FUNCTION_BLOCK PUBLIC ACMethodMixing EXTENDS ACMethodRouteBase
VAR_INPUT
END_VAR
VAR_OUTPUT
END_VAR
VAR PERSISTENT
	_Parameter : ACMethodMixingP;
	_Result : ACMethodMixingR;
END_VAR

PROPERTY IsValid : BOOL
GET
IsValid := TRUE;
END_GET
END_PROPERTY

PROPERTY Parameter : ACMethodMixingP
GET
Parameter := _Parameter;
END_GET
SET // PUBLIC
_Parameter := Parameter;
END_SET
END_PROPERTY

PROPERTY Result : ACMethodMixingR
GET
Result := _Result;
END_GET
SET // PUBLIC
_Result := Result;
END_SET
END_PROPERTY

END_FUNCTION_BLOCK

(* stored: Version 1.1.0.1, ProductVersion 3.1.4022.7
   POU ACMethodMixing: Id {e34540a1-26ae-4e11-859a-e6bce4e16774}, SpecialFunc None
   Property IsValid: Id {42f4db85-f64f-43b4-97a5-718885284ed0}
   Get Get: Id {b18a4950-feb2-491e-becd-006bc04d95b6}
   Property Parameter: Id {b7128a30-ff08-4a6d-ba85-4974fbf3f524}
   Get Get: Id {046d3d49-095b-4ae6-975c-499e718bc5b5}
   Set Set: Id {2532546b-7ad8-4f0c-90d7-f35a83733087}
   Property Result: Id {8ddda802-b4e1-41a9-bee9-a82d418e5a74}
   Get Get: Id {5425cf10-1e16-4355-8b91-1ae8a13849bd}
   Set Set: Id {90ab7058-3e29-4c68-9abb-c086e958cd38} *)
